ABB RobotStudio station: Solution_3_Template.rspag

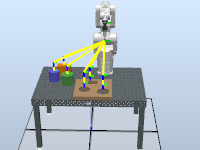
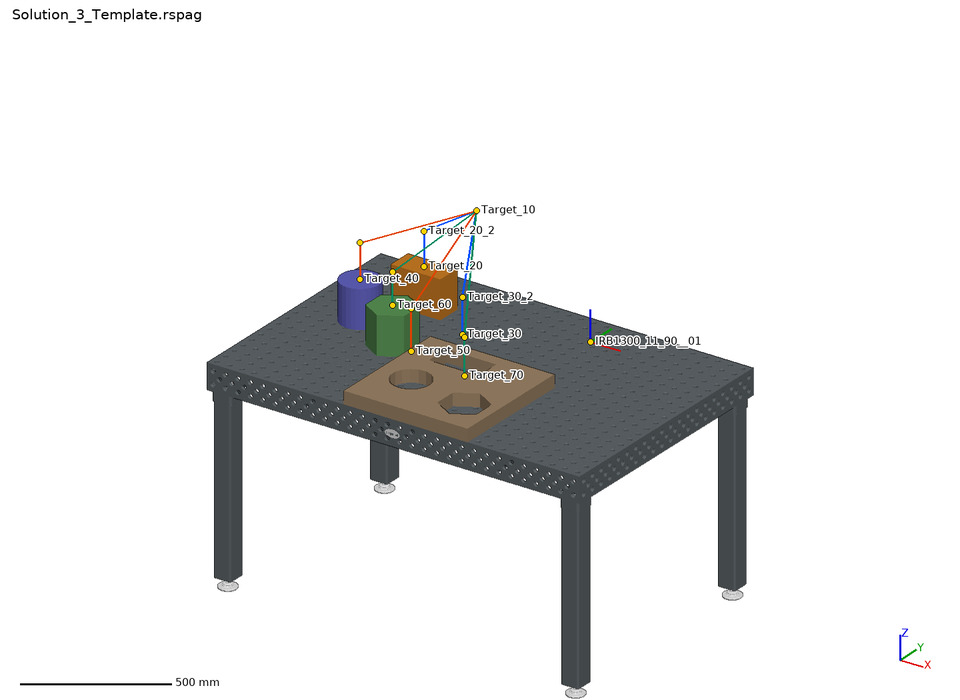
[picture v1: parts stored in the station drawn from their meshes, with robot base, taught points and paths (robot models come from the ABB library and are not in the file)]
--- station ---
Station Solution_1_Tutorial (saved by RobotStudio 21.4.9700.0)
Controller Controller1, task T_ROB1: task frame (RAPID world) sits at (200, 350, 830) mm, rotated rx 0 ry 0 rz -90 deg in the station
Controller Controller1
  mechanical unit ROB_1: IRB1300_11_90__01, 6 joints, base frame (0, 0, 0) mm
Layout (positions relative to the parent item):
  - table [part] at (-200, -500, 830) mm, size 500 x 500 x 50 mm
  - object_1 [part] at (-600, -150, 830) mm, size 200 x 100 x 150 mm
  - object_2 [part] at (-650, -150, 830) mm, size 149.5 x 149.7 x 150 mm
  - object_3 [part] at (-700, -200, 830) mm, size 155.5 x 179.5 x 150 mm
  - siegmund_1500_1000 [part], size 1500 x 1010.3 x 830 mm
  - object_11 [part] at (-200, -500, 830) mm, size 200 x 100 x 150 mm
  - object_22 [part] at (-200, -500, 830) mm, size 149.5 x 149.7 x 150 mm
  - object_33 [part] at (-200, -500, 830) mm, size 155.5 x 179.5 x 150 mm
  - IRB1300_11_90__01 [mechanism, from Robots\IRB1300_11_90__01.rslib] at (200, 350, 830) mm, rotated rx 0 ry 0 rz -90 deg; joint values [0, 0, 0, 0, 0.8727, 0] (rad or m)
  - MyTool [mechanism, from Training Objects\myTool.rslib] at (200, -182.85, 1770.06) mm, rotated rx 180 ry 40 rz 90 deg
  - Positioner_obj_1 [smart component, from Components\Positioner.rslib]
      properties: Object=object_1; Position=[-0.6 -0.15 0.83]; Orientation=[0 0 0]; Reference=Global; ReferenceObject=(none)
  - Positioner_obj_2 [smart component, from Components\Positioner.rslib]
      properties: Object=object_2; Position=[-0.65 -0.15 0.83]; Orientation=[0 0 0]; Reference=Global; ReferenceObject=(none)
  - Positioner_obj_3 [smart component, from Components\Positioner.rslib]
      properties: Object=object_3; Position=[-0.7 -0.2 0.83]; Orientation=[0 0 0]; Reference=Global; ReferenceObject=(none)
  - Attacher_obj_1 [smart component, from Components\Attacher.rslib]
      properties: Parent=MyTool; Flange=0; Child=object_1; Mount=false; Offset=[0 0 0]; Orientation=[0 0 0]
  - Attacher_obj_2 [smart component, from Components\Attacher.rslib]
      properties: Parent=MyTool; Flange=0; Child=object_2; Mount=false; Offset=[0 0 0]; Orientation=[0 0 0]
  - Attacher_obj_3 [smart component, from Components\Attacher.rslib]
      properties: Parent=MyTool; Flange=0; Child=object_3; Mount=false; Offset=[0 0 0]; Orientation=[0 0 0]
  - Detacher_obj_1 [smart component, from Components\Detacher.rslib]
      properties: Child=object_1; KeepPosition=true
  - Detacher_obj_2 [smart component, from Components\Detacher.rslib]
      properties: Child=object_2; KeepPosition=true
  - Detacher_obj_3 [smart component, from Components\Detacher.rslib]
      properties: Child=object_3; KeepPosition=true
Attachment: MyTool is attached to IRB1300_11_90__01 / Link6
Station signals: DI object_1_positioner, DI object_2_positioner, DI object_3_positioner
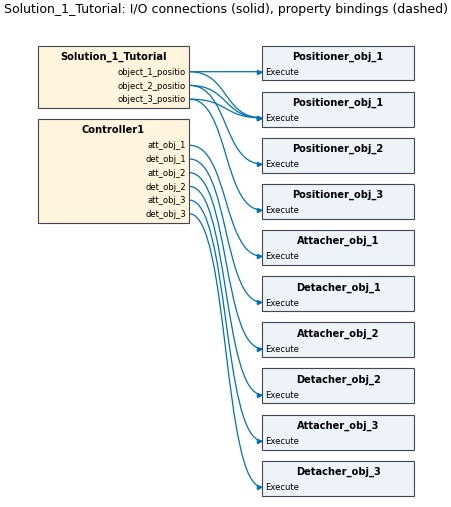
Station logic (signal -> signal, property => property):
  Solution_1_Tutorial.object_1_positioner -> Positioner_obj_1.Execute
  Solution_1_Tutorial.object_2_positioner -> Positioner_obj_2.Execute
  Solution_1_Tutorial.object_3_positioner -> Positioner_obj_3.Execute
  Solution_1_Tutorial.object_1_positioner -> Positioner_obj_1.Execute
  Solution_1_Tutorial.object_2_positioner -> Positioner_obj_2.Execute
  Solution_1_Tutorial.object_3_positioner -> Positioner_obj_3.Execute
  Controller1.att_obj_1 -> Attacher_obj_1.Execute
  Controller1.det_obj_1 -> Detacher_obj_1.Execute
  Controller1.att_obj_2 -> Attacher_obj_2.Execute
  Controller1.det_obj_2 -> Detacher_obj_2.Execute
  Controller1.att_obj_3 -> Attacher_obj_3.Execute
  Controller1.det_obj_3 -> Detacher_obj_3.Execute

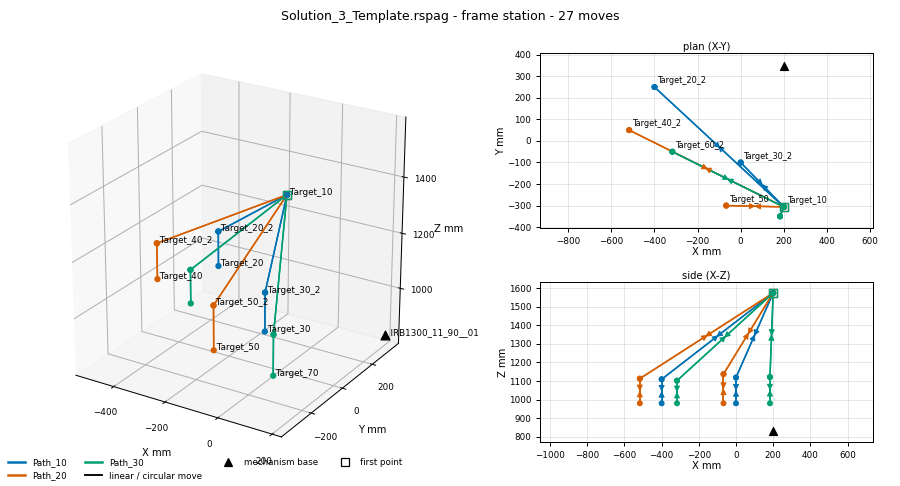
[picture p0: tool path of Solution_3_Template.rspag in frame station, 27 of 27 moves have a stored position in this frame; points joined in program order, loops and branches not executed]
--- Backups/Controller1/RAPID/TASK1/PROGMOD/CalibData.modx ---
MODULE CalibData
    PERS tooldata MyTool:=[TRUE,[[31.792631019,0,229.638935148],[0.945518576,0,0.325568154,0]],[1,[0,0,1],[1,0,0,0],0,0,0]];
ENDMODULE

--- Backups/Controller1/RAPID/TASK1/PROGMOD/Module1.modx ---
MODULE Module1
        CONST robtarget Target_10:=[[656.105378762,0,743.706460627],[0.017452407,0,0.999847695,0],[-1,0,-1,0],[9E+09,9E+09,9E+09,9E+09,9E+09,9E+09]];
    CONST robtarget Target_20_2:=[[100,-600,279.251353636],[0.017452407,0,0.999847695,0],[-2,0,-2,0],[9E+09,9E+09,9E+09,9E+09,9E+09,9E+09]];
    CONST robtarget Target_20:=[[100,-600,150],[0.017452407,0,0.999847695,0],[-2,0,-2,0],[9E+09,9E+09,9E+09,9E+09,9E+09,9E+09]];
    CONST robtarget Target_30_2:=[[450,-200,288.692856548],[0.017452407,0,0.999847695,0],[-1,1,-2,0],[9E+09,9E+09,9E+09,9E+09,9E+09,9E+09]];
    CONST robtarget Target_30:=[[450,-200,150],[0.017452407,0,0.999847695,0],[-1,1,-3,0],[9E+09,9E+09,9E+09,9E+09,9E+09,9E+09]];
    CONST robtarget Target_40_2:=[[300,-717.298,282.774630166],[0.017452407,0,0.999847695,0],[-1,0,-2,0],[9E+09,9E+09,9E+09,9E+09,9E+09,9E+09]];
    CONST robtarget Target_40:=[[300,-717.298,150],[0.017452407,0,0.999847695,0],[-1,0,-2,0],[9E+09,9E+09,9E+09,9E+09,9E+09,9E+09]];
    CONST robtarget Target_50_2:=[[650,-267.298,307.067020555],[0.017452407,0,0.999847695,0],[-1,1,-2,0],[9E+09,9E+09,9E+09,9E+09,9E+09,9E+09]];
    CONST robtarget Target_50:=[[650,-267.298,150],[0.017452407,0,0.999847695,0],[-1,1,-2,0],[9E+09,9E+09,9E+09,9E+09,9E+09,9E+09]];
    CONST robtarget Target_60_2:=[[400,-517.298,271.901920667],[0.017452407,0,0.999847695,0],[-1,0,-2,0],[9E+09,9E+09,9E+09,9E+09,9E+09,9E+09]];
    CONST robtarget Target_60:=[[400,-517.298,150],[0.017452407,0,0.999847695,0],[-1,0,-2,0],[9E+09,9E+09,9E+09,9E+09,9E+09,9E+09]];
    CONST robtarget Target_70_2:=[[700,-17.298,291.51943135],[0.017452407,0,0.999847695,0],[-1,1,-2,0],[9E+09,9E+09,9E+09,9E+09,9E+09,9E+09]];
    CONST robtarget Target_70:=[[700,-17.298,150],[0.017452407,0,0.999847695,0],[-1,1,-2,0],[9E+09,9E+09,9E+09,9E+09,9E+09,9E+09]];

    PROC main()
        ! Pick object 3
        Path_30;
        ! Pick object 2
        Path_20;
        ! Pick object 1
        Path_10;
    ENDPROC
    PROC Path_10()
        MoveL Target_10,v150,fine,MyTool\WObj:=wobj0;
        MoveL Target_20_2,v150,fine,MyTool\WObj:=wobj0;
        MoveL Target_20,v150,fine,MyTool\WObj:=wobj0;
        PulseDO att_obj_1;
        WaitTime 0.5;
        MoveL Target_20_2,v150,fine,MyTool\WObj:=wobj0;
        MoveL Target_10,v150,fine,MyTool\WObj:=wobj0;
        MoveL Target_30_2,v150,fine,MyTool\WObj:=wobj0;
        MoveL Target_30,v150,fine,MyTool\WObj:=wobj0;
        PulseDO det_obj_1;
        WaitTime 0.5;
        MoveL Target_30_2,v150,fine,MyTool\WObj:=wobj0;
        MoveL Target_10,v150,fine,MyTool\WObj:=wobj0;
    ENDPROC
    PROC Path_20()
        MoveL Target_10,v150,fine,MyTool\WObj:=wobj0;
        MoveL Target_40_2,v150,fine,MyTool\WObj:=wobj0;
        MoveL Target_40,v150,fine,MyTool\WObj:=wobj0;
        PulseDO att_obj_2;
        WaitTime 0.5;
        MoveL Target_40_2,v150,fine,MyTool\WObj:=wobj0;
        MoveL Target_10,v150,fine,MyTool\WObj:=wobj0;
        MoveL Target_50_2,v150,fine,MyTool\WObj:=wobj0;
        MoveL Target_50,v150,fine,MyTool\WObj:=wobj0;
        PulseDO det_obj_2;
        WaitTime 0.5;
        MoveL Target_50_2,v150,fine,MyTool\WObj:=wobj0;
        MoveL Target_10,v150,fine,MyTool\WObj:=wobj0;
    ENDPROC
    PROC Path_30()
        MoveL Target_10,v150,fine,MyTool\WObj:=wobj0;
        MoveL Target_60_2,v150,fine,MyTool\WObj:=wobj0;
        MoveL Target_60,v150,fine,MyTool\WObj:=wobj0;
        PulseDO att_obj_3;
        WaitTime 0.5;
        MoveL Target_60_2,v150,fine,MyTool\WObj:=wobj0;
        MoveL Target_10,v150,fine,MyTool\WObj:=wobj0;
        MoveL Target_70_2,v150,fine,MyTool\WObj:=wobj0;
        MoveL Target_70,v150,fine,MyTool\WObj:=wobj0;
        PulseDO det_obj_3;
        WaitTime 0.5;
        MoveL Target_70_2,v150,fine,MyTool\WObj:=wobj0;
        MoveL Target_10,v150,fine,MyTool\WObj:=wobj0;
    ENDPROC
ENDMODULE

--- Backups/Controller1/SYSPAR/EIO.cfg ---
EIO:CFG_1.0:7:0::
#
EIO_SIGNAL:

      -Name "att_obj_1" -SignalType "DO"

      -Name "att_obj_2" -SignalType "DO"

      -Name "att_obj_3" -SignalType "DO"

      -Name "det_obj_1" -SignalType "DO"

      -Name "det_obj_2" -SignalType "DO"

      -Name "det_obj_3" -SignalType "DO"

#CTRL_SIGNATURE:oe8ag/ugcV6aFXzoXZRUOm/9jxLYrMI2DDKuB3P1nqcO9WXIrW/iqCi3Tn8xI77GZMSes/d02tvYviDtgJmK9g==

--- Backups/Controller1/SYSPAR/PROC.cfg ---
PROC:CFG_1.0:7:0::

#CTRL_SIGNATURE:I+y2QaV15gWtHGM+5Z4idi3NiusZu29hLyokxM3ohwogLM8MfydOTWOtI2G6szFitByh5svEYsXD7agPogo+dQ==
